FUNCTION_BLOCK C90_FB_PackCodeGenerator

VAR_INPUT
	bStart:BOOL;
	nPackCodeLenght:INT;
END_VAR

VAR_OUTPUT
	sPackCode:T_PACK_Barcode;
END_VAR

VAR
	sAsciiSymbol:STRING(1);
	nIndex:INT;
	fbPackCharacterGenerator:C90_FB_CharacterGenerator;
END_VAR

(*Pack code generator *********************************************************************)
	IF NOT bStart THEN
		sPackCode:='';
	END_IF

	FOR nIndex:=1 TO nPackCodeLenght DO

		fbPackCharacterGenerator	(
									nMinAsciiRange:=16#21,
									nMaxAsciiRange:=16#7A,
									sAsciiSymbol=>sAsciiSymbol
								);

		(*Pack string creator*)
		sPackCode:=CONCAT(sPackCode, sAsciiSymbol);

	END_FOR

END_FUNCTION_BLOCK

(* stored: Version 1.1.0.1, ProductVersion 3.1.4024.15
   POU C90_FB_PackCodeGenerator: Id {5a7dae56-17fc-4c84-bd4d-95b4ed4d90a2}, SpecialFunc None *)
